FUNCTION_BLOCK Section6Ctrl (* Basic Function Block Type *)
  (* Standard: 61499-2 *)
  (* Version 0.0, 5/28/2018, taavi, nxtControl GmbH, Template *)
  PACKAGE Main;
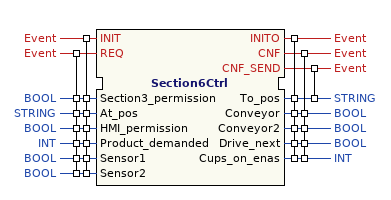
  EVENT_INPUT
    INIT WITH Section3_permission, At_pos, HMI_permission, Product_demanded, Sensor1, Sensor2; (* Initialization Request *)
    REQ WITH Section3_permission, At_pos, HMI_permission, Product_demanded, Sensor1, Sensor2; (* Normal Execution Request *)
  END_EVENT
  EVENT_OUTPUT
    INITO WITH To_pos, Conveyor, Conveyor2, Drive_next, Cups_on_enas; (* Initialization Confirm *)
    CNF WITH Conveyor, Conveyor2, Drive_next, Cups_on_enas; (* Execution Confirmation *)
    CNF_SEND WITH To_pos;
  END_EVENT
  VAR_INPUT
    Section3_permission : BOOL; (* Input event qualifier *)
    At_pos : STRING;
    HMI_permission : BOOL;
    Product_demanded : INT;
    Sensor1 : BOOL;
    Sensor2 : BOOL;
  END_VAR
  VAR_OUTPUT
    To_pos : STRING; (* Output event qualifier *)
    Conveyor : BOOL;
    Conveyor2 : BOOL;
    Drive_next : BOOL;
    Cups_on_enas : INT;
  END_VAR
  VAR
    Product_to_collect : INT;
    Cups_to_deliver : INT;
    Cups_on_enas_internal : INT;
    TimeStamp : DATE_AND_TIME;
  END_VAR
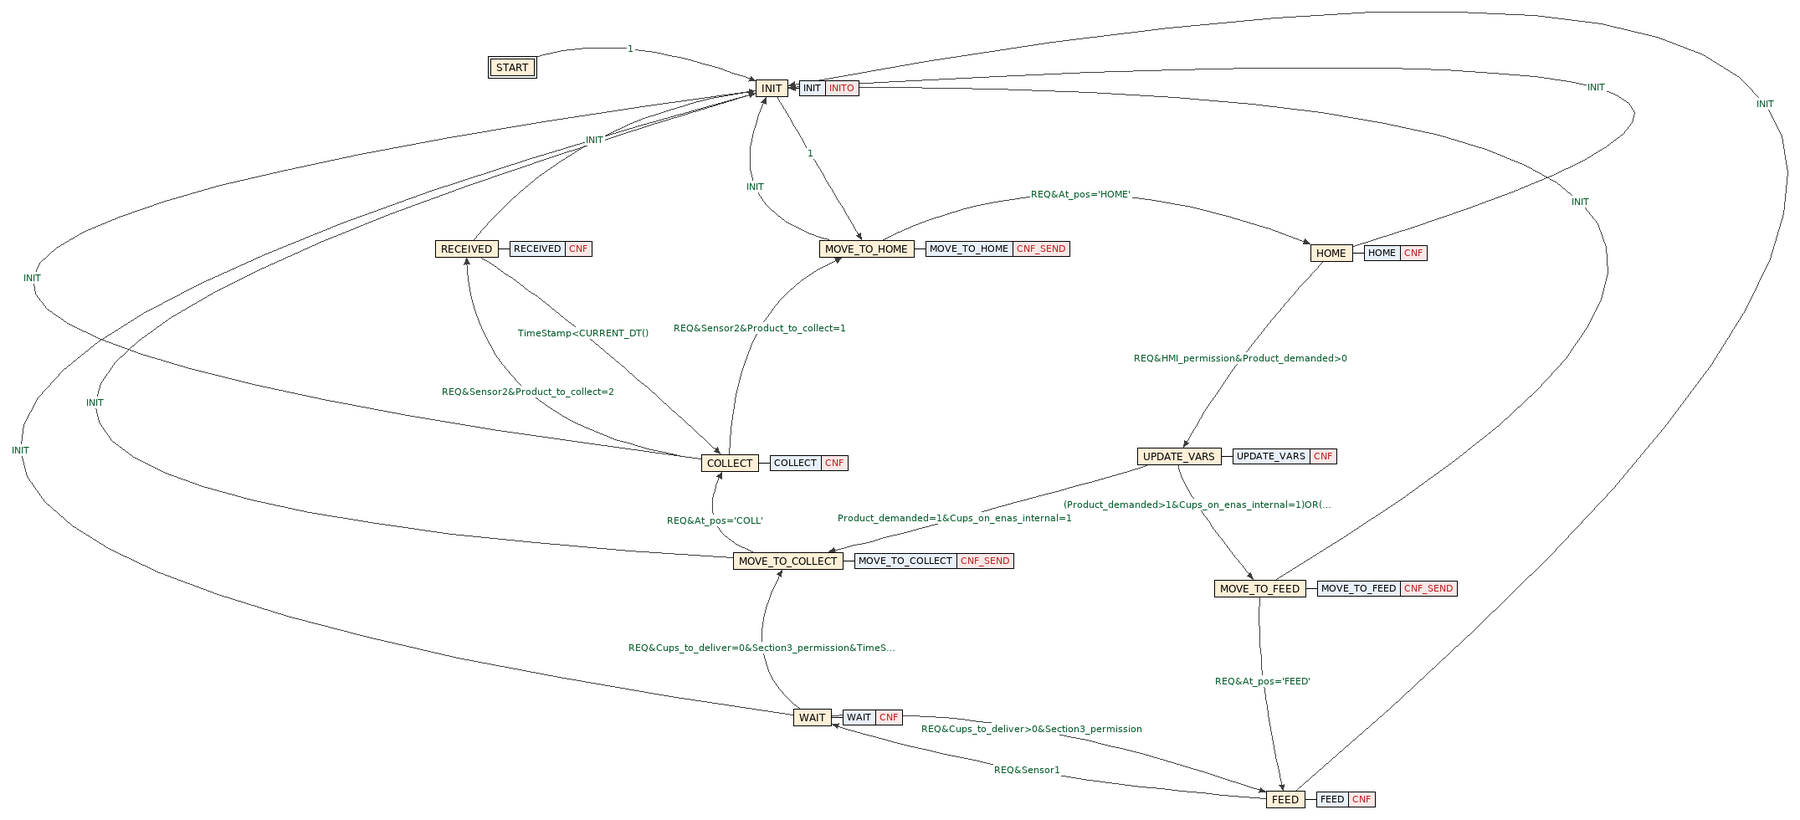
  EC_STATES
    START; (* Initial State *)
    INIT : INIT -> INITO; (* Initialization *)
    MOVE_TO_HOME : MOVE_TO_HOME -> CNF_SEND;
    HOME : HOME -> CNF;
    RECEIVED : RECEIVED -> CNF;
    COLLECT : COLLECT -> CNF;
    UPDATE_VARS : UPDATE_VARS -> CNF;
    MOVE_TO_COLLECT : MOVE_TO_COLLECT -> CNF_SEND;
    MOVE_TO_FEED : MOVE_TO_FEED -> CNF_SEND;
    WAIT : WAIT -> CNF;
    FEED : FEED -> CNF;
  END_STATES
  EC_TRANSITIONS
    START TO INIT := 1;
    INIT TO MOVE_TO_HOME := 1;
    COLLECT TO RECEIVED := REQ&Sensor2&Product_to_collect=2;
    RECEIVED TO COLLECT := TimeStamp<CURRENT_DT();
    MOVE_TO_HOME TO HOME := REQ&At_pos='HOME';
    HOME TO UPDATE_VARS := REQ&HMI_permission&Product_demanded>0;
    MOVE_TO_FEED TO FEED := REQ&At_pos='FEED';
    FEED TO WAIT := REQ&Sensor1;
    WAIT TO FEED := REQ&Cups_to_deliver>0&Section3_permission;
    WAIT TO MOVE_TO_COLLECT := REQ&Cups_to_deliver=0&Section3_permission&TimeStamp<CURRENT_DT();
    MOVE_TO_COLLECT TO COLLECT := REQ&At_pos='COLL';
    UPDATE_VARS TO MOVE_TO_COLLECT := Product_demanded=1&Cups_on_enas_internal=1;
    UPDATE_VARS TO MOVE_TO_FEED := (Product_demanded>1&Cups_on_enas_internal=1)OR(Product_demanded>=1&Cups_on_enas_internal=0);
    COLLECT TO MOVE_TO_HOME := REQ&Sensor2&Product_to_collect=1;
    HOME TO INIT := INIT;
    MOVE_TO_HOME TO INIT := INIT;
    RECEIVED TO INIT := INIT;
    COLLECT TO INIT := INIT;
    MOVE_TO_COLLECT TO INIT := INIT;
    MOVE_TO_FEED TO INIT := INIT;
    FEED TO INIT := INIT;
    WAIT TO INIT := INIT;
  END_TRANSITIONS
  ALGORITHM INIT IN ST: (* Initialization algorithm *)
;
Conveyor := FALSE;
To_pos := 'NONE';
Drive_next := FALSE;
Product_to_collect := 0;
Cups_to_deliver := 0;
Cups_on_enas := 0;
Cups_on_enas_internal := 0;
  END_ALGORITHM
  ALGORITHM REQ IN ST: (* Normally executed algorithm *)
;
  END_ALGORITHM
  ALGORITHM MOVE_TO_HOME IN ST:
;
Conveyor := FALSE;
To_pos := 'HOME';
Drive_next := FALSE;
Product_to_collect := 0;
Cups_on_enas := Cups_on_enas_internal;
  END_ALGORITHM
  ALGORITHM RECEIVED IN ST:
;
To_pos := 'NONE';
Conveyor := TRUE;
Product_to_collect := Product_to_collect - 1;
Drive_next := TRUE;
TimeStamp := ADD_DT_TIME(CURRENT_DT(),T#2.0s);
  END_ALGORITHM
  ALGORITHM HOME IN ST:
;
Conveyor := FALSE;
To_pos := 'NONE';
Drive_next := FALSE;
Cups_on_enas := Cups_on_enas_internal;
  END_ALGORITHM
  ALGORITHM COLLECT IN ST:
;
To_pos := 'NONE';
Conveyor2 := TRUE;
Drive_next := FALSE;
Cups_on_enas := Cups_on_enas_internal;
  END_ALGORITHM
  ALGORITHM UPDATE_VARS IN ST:
;

IF Product_demanded >= 2 THEN
	Product_to_collect := 2;
ELSE
	Product_to_collect := 1;
END_IF;

IF Cups_on_enas_internal = 1 THEN
	Cups_to_deliver := 1;
ELSE
  Cups_to_deliver := 2;
END_IF;

IF Cups_on_enas_internal = 1 & Product_demanded = 1 THEN
	Cups_to_deliver := 0;
END_IF;
  END_ALGORITHM
  ALGORITHM MOVE_TO_COLLECT IN ST:
;
Conveyor := FALSE;
To_pos := 'COLL';
IF Cups_on_enas_internal = 1 THEN Drive_next := TRUE;
ELSE Drive_next := FALSE;
END_IF;
  END_ALGORITHM
  ALGORITHM MOVE_TO_FEED IN ST:
;
Conveyor := FALSE;
To_pos := 'FEED';
Drive_next := FALSE;
Cups_on_enas := Cups_on_enas_internal;
  END_ALGORITHM
  ALGORITHM WAIT IN ST:
;
To_pos := 'NONE';
Conveyor := FALSE;
Drive_next := FALSE;
Cups_to_deliver := Cups_to_deliver - 1;
Cups_on_enas := Cups_on_enas_internal + 1;
Cups_on_enas_internal := Cups_on_enas_internal + 1;
TimeStamp := ADD_DT_TIME(CURRENT_DT(),T#1.0s);
  END_ALGORITHM
  ALGORITHM FEED IN ST:
;
To_pos := 'NONE';
Conveyor := TRUE;
Drive_next := FALSE;
Cups_on_enas := Cups_on_enas_internal;
  END_ALGORITHM
END_FUNCTION_BLOCK
